Xinje XDPPro project, PLC1: XD3-32 (software 3.7.14 2021-12-24)

PROGRAM 梯形图

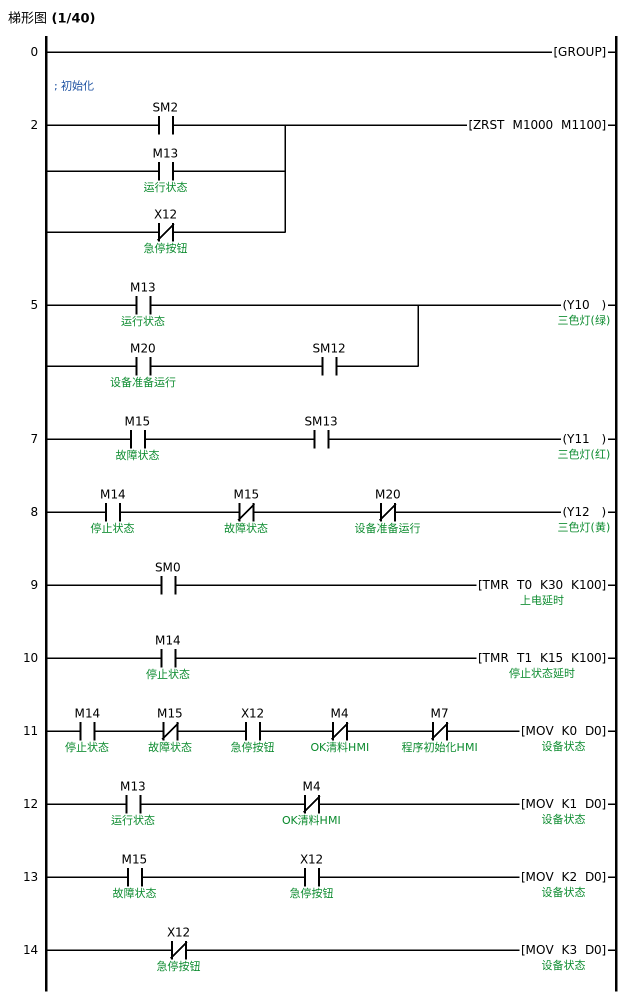
GROUP
; 初始化
LD     SM2
OR     M13	; 运行状态
ORI    X12	; 急停按钮
ZRST   M1000 M1100
LD     M13	; 运行状态
LD     M20	; 设备准备运行
AND    SM12
ORB
OUT    Y10	; 三色灯(绿)
LD     M15	; 故障状态
AND    SM13
OUT    Y11	; 三色灯(红)
LD     M14	; 停止状态
ANI    M15	; 故障状态
ANI    M20	; 设备准备运行
OUT    Y12	; 三色灯(黄)
LD     SM0
TMR    T0 K30 K100	; 上电延时
LD     M14	; 停止状态
TMR    T1 K15 K100	; 停止状态延时
LD     M14	; 停止状态
ANI    M15	; 故障状态
AND    X12	; 急停按钮
ANI    M4	; OK清料HMI
ANI    M7	; 程序初始化HMI
MOV    K0 D0	; 设备状态
LD     M13	; 运行状态
ANI    M4	; OK清料HMI
MOV    K1 D0	; 设备状态
LD     M15	; 故障状态
AND    X12	; 急停按钮
MOV    K2 D0	; 设备状态
LDI    X12	; 急停按钮
MOV    K3 D0	; 设备状态

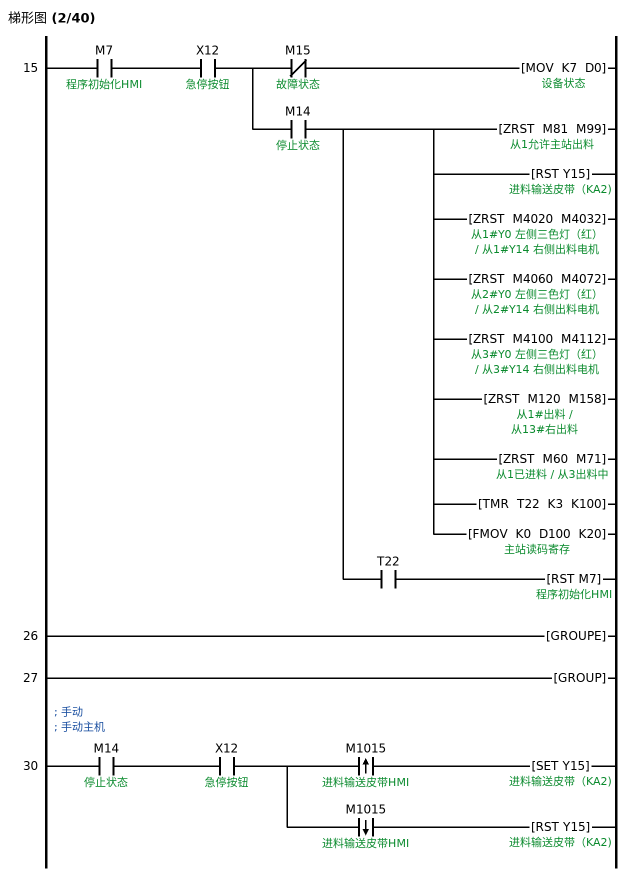
LD     M7	; 程序初始化HMI
AND    X12	; 急停按钮
MPS
ANI    M15	; 故障状态
MOV    K7 D0	; 设备状态
MPP
AND    M14	; 停止状态
ZRST   M81 M99	; 从1允许主站出料
RST    Y15	; 进料输送皮带（KA2)
ZRST   M4020 M4032	; 从1#Y0 左侧三色灯（红） / 从1#Y14 右侧出料电机
ZRST   M4060 M4072	; 从2#Y0 左侧三色灯（红） / 从2#Y14 右侧出料电机
ZRST   M4100 M4112	; 从3#Y0 左侧三色灯（红） / 从3#Y14 右侧出料电机
ZRST   M120 M158	; 从1#出料 / 从13#右出料
ZRST   M60 M71	; 从1已进料 / 从3出料中
TMR    T22 K3 K100
FMOV   K0 D100 K20	; 主站读码寄存
AND    T22
RST    M7	; 程序初始化HMI
GROUPE
GROUP
; 手动
; 手动主机
LD     M14	; 停止状态
AND    X12	; 急停按钮
MPS
ANDP   M1015	; 进料输送皮带HMI
SET    Y15	; 进料输送皮带（KA2)
MPP
ANDF   M1015	; 进料输送皮带HMI
RST    Y15	; 进料输送皮带（KA2)

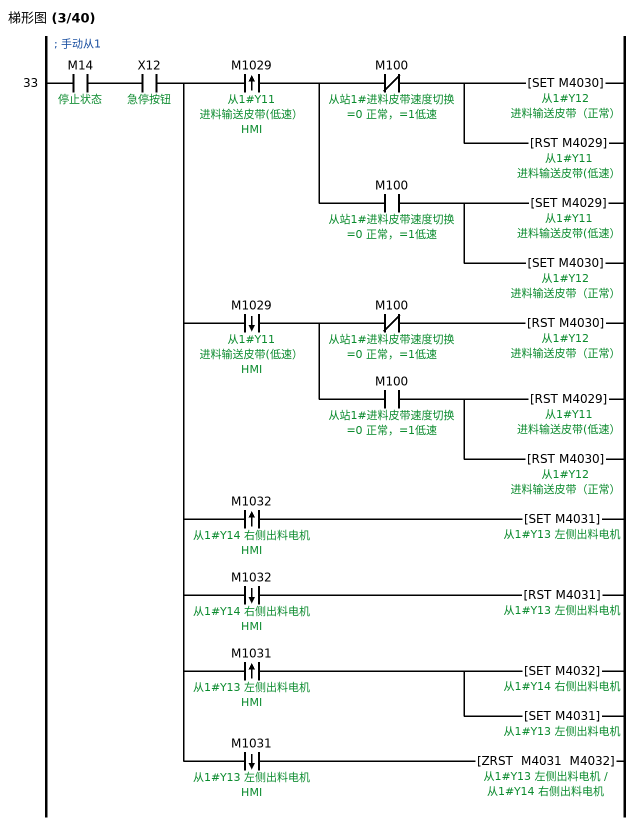
; 手动从1
LD     M14	; 停止状态
AND    X12	; 急停按钮
MPS
ANDP   M1029	; 从1#Y11 进料输送皮带(低速）       HMI
MPS
ANI    M100	; 从站1#进料皮带速度切换=0 正常，=1低速
SET    M4030	; 从1#Y12 进料输送皮带（正常）
RST    M4029	; 从1#Y11 进料输送皮带(低速）
MPP
AND    M100	; 从站1#进料皮带速度切换=0 正常，=1低速
SET    M4029	; 从1#Y11 进料输送皮带(低速）
SET    M4030	; 从1#Y12 进料输送皮带（正常）
MRD
ANDF   M1029	; 从1#Y11 进料输送皮带(低速）       HMI
MPS
ANI    M100	; 从站1#进料皮带速度切换=0 正常，=1低速
RST    M4030	; 从1#Y12 进料输送皮带（正常）
MPP
AND    M100	; 从站1#进料皮带速度切换=0 正常，=1低速
RST    M4029	; 从1#Y11 进料输送皮带(低速）
RST    M4030	; 从1#Y12 进料输送皮带（正常）
MRD
ANDP   M1032	; 从1#Y14 右侧出料电机       HMI
SET    M4031	; 从1#Y13 左侧出料电机
MRD
ANDF   M1032	; 从1#Y14 右侧出料电机       HMI
RST    M4031	; 从1#Y13 左侧出料电机
MRD
ANDP   M1031	; 从1#Y13 左侧出料电机       HMI
SET    M4032	; 从1#Y14 右侧出料电机
SET    M4031	; 从1#Y13 左侧出料电机
MPP
ANDF   M1031	; 从1#Y13 左侧出料电机       HMI
ZRST   M4031 M4032	; 从1#Y13 左侧出料电机 / 从1#Y14 右侧出料电机

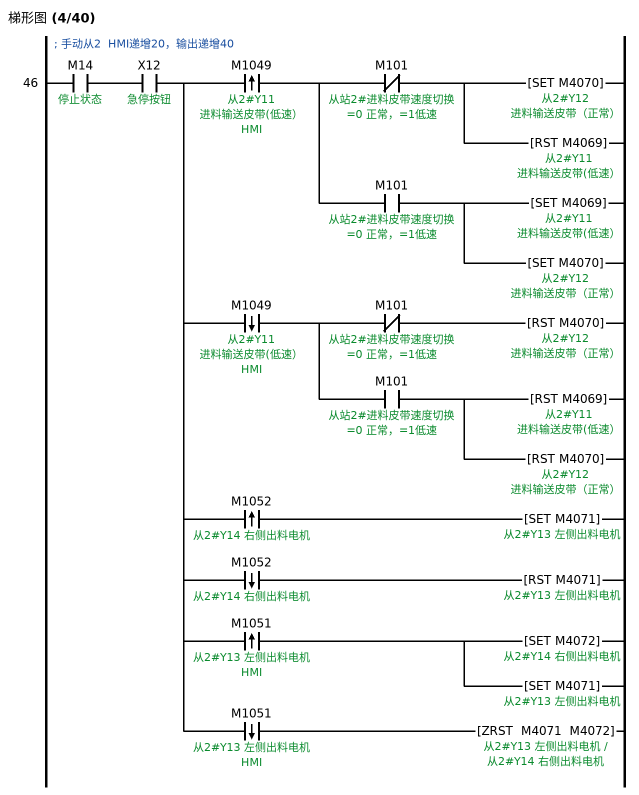
; 手动从2  HMI递增20，输出递增40
LD     M14	; 停止状态
AND    X12	; 急停按钮
MPS
ANDP   M1049	; 从2#Y11 进料输送皮带(低速）       HMI
MPS
ANI    M101	; 从站2#进料皮带速度切换=0 正常，=1低速
SET    M4070	; 从2#Y12 进料输送皮带（正常）
RST    M4069	; 从2#Y11 进料输送皮带(低速）
MPP
AND    M101	; 从站2#进料皮带速度切换=0 正常，=1低速
SET    M4069	; 从2#Y11 进料输送皮带(低速）
SET    M4070	; 从2#Y12 进料输送皮带（正常）
MRD
ANDF   M1049	; 从2#Y11 进料输送皮带(低速）       HMI
MPS
ANI    M101	; 从站2#进料皮带速度切换=0 正常，=1低速
RST    M4070	; 从2#Y12 进料输送皮带（正常）
MPP
AND    M101	; 从站2#进料皮带速度切换=0 正常，=1低速
RST    M4069	; 从2#Y11 进料输送皮带(低速）
RST    M4070	; 从2#Y12 进料输送皮带（正常）
MRD
ANDP   M1052	; 从2#Y14 右侧出料电机
SET    M4071	; 从2#Y13 左侧出料电机
MRD
ANDF   M1052	; 从2#Y14 右侧出料电机
RST    M4071	; 从2#Y13 左侧出料电机
MRD
ANDP   M1051	; 从2#Y13 左侧出料电机       HMI
SET    M4072	; 从2#Y14 右侧出料电机
SET    M4071	; 从2#Y13 左侧出料电机
MPP
ANDF   M1051	; 从2#Y13 左侧出料电机       HMI
ZRST   M4071 M4072	; 从2#Y13 左侧出料电机 / 从2#Y14 右侧出料电机

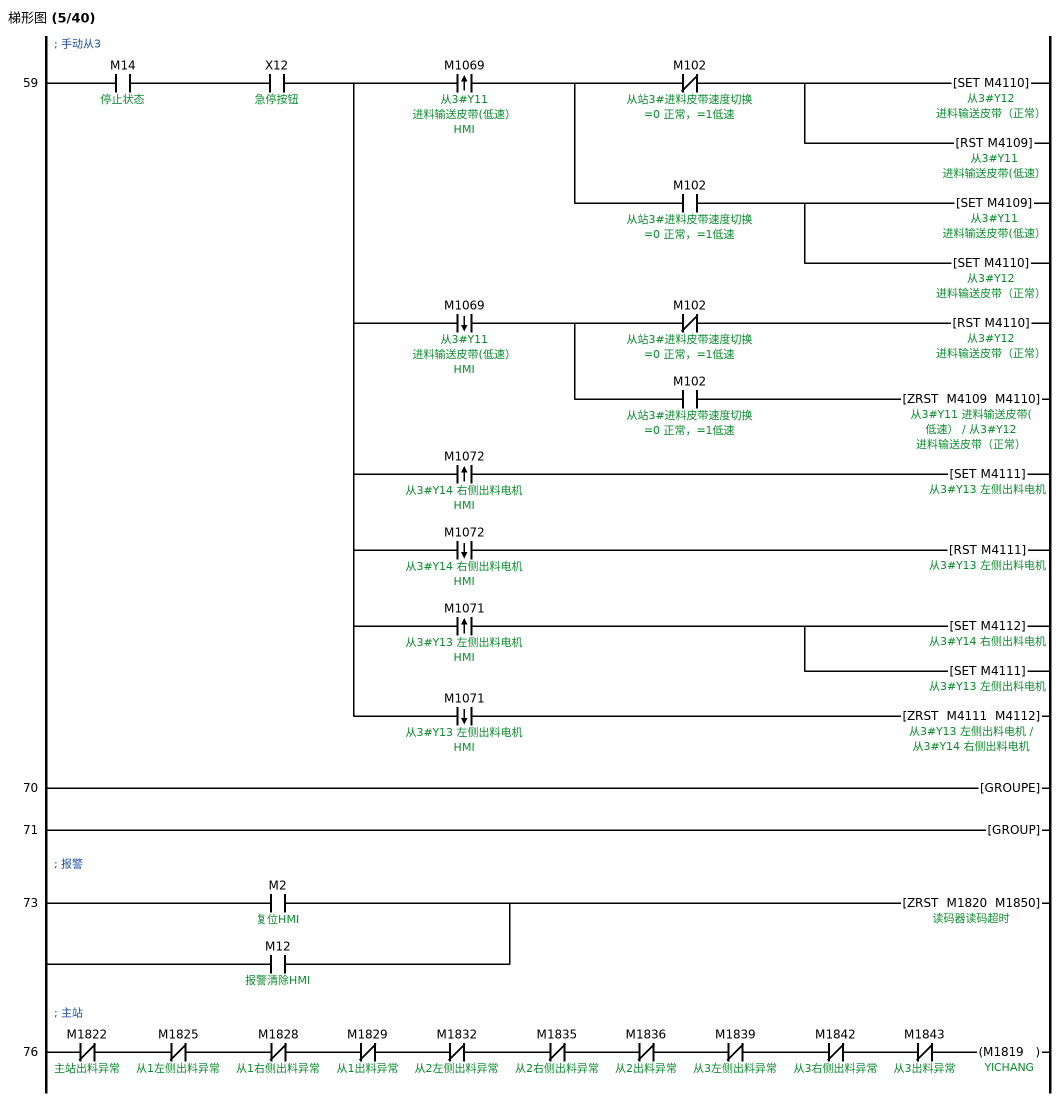
; 手动从3
LD     M14	; 停止状态
AND    X12	; 急停按钮
MPS
ANDP   M1069	; 从3#Y11 进料输送皮带(低速）       HMI
MPS
ANI    M102	; 从站3#进料皮带速度切换=0 正常，=1低速
SET    M4110	; 从3#Y12 进料输送皮带（正常）
RST    M4109	; 从3#Y11 进料输送皮带(低速）
MPP
AND    M102	; 从站3#进料皮带速度切换=0 正常，=1低速
SET    M4109	; 从3#Y11 进料输送皮带(低速）
SET    M4110	; 从3#Y12 进料输送皮带（正常）
MRD
ANDF   M1069	; 从3#Y11 进料输送皮带(低速）       HMI
MPS
ANI    M102	; 从站3#进料皮带速度切换=0 正常，=1低速
RST    M4110	; 从3#Y12 进料输送皮带（正常）
MPP
AND    M102	; 从站3#进料皮带速度切换=0 正常，=1低速
ZRST   M4109 M4110	; 从3#Y11 进料输送皮带(低速） / 从3#Y12 进料输送皮带（正常）
MRD
ANDP   M1072	; 从3#Y14 右侧出料电机       HMI
SET    M4111	; 从3#Y13 左侧出料电机
MRD
ANDF   M1072	; 从3#Y14 右侧出料电机       HMI
RST    M4111	; 从3#Y13 左侧出料电机
MRD
ANDP   M1071	; 从3#Y13 左侧出料电机       HMI
SET    M4112	; 从3#Y14 右侧出料电机
SET    M4111	; 从3#Y13 左侧出料电机
MPP
ANDF   M1071	; 从3#Y13 左侧出料电机       HMI
ZRST   M4111 M4112	; 从3#Y13 左侧出料电机 / 从3#Y14 右侧出料电机
GROUPE
GROUP
; 报警
LD     M2	; 复位HMI
OR     M12	; 报警清除HMI
ZRST   M1820 M1850	; 读码器读码超时
; 主站
LDI    M1822	; 主站出料异常
ANI    M1825	; 从1左侧出料异常
ANI    M1828	; 从1右侧出料异常
ANI    M1829	; 从1出料异常
ANI    M1832	; 从2左侧出料异常
ANI    M1835	; 从2右侧出料异常
ANI    M1836	; 从2出料异常
ANI    M1839	; 从3左侧出料异常
ANI    M1842	; 从3右侧出料异常
ANI    M1843	; 从3出料异常
OUT    M1819	; YICHANG

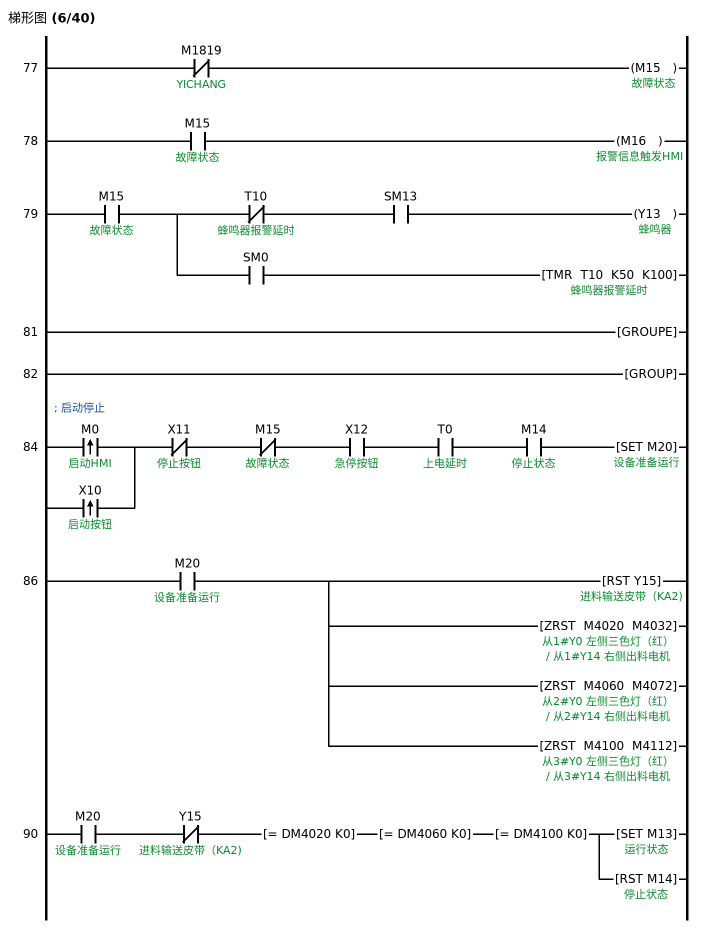
LDI    M1819	; YICHANG
OUT    M15	; 故障状态
LD     M15	; 故障状态
OUT    M16	; 报警信息触发HMI
LD     M15	; 故障状态
MPS
ANI    T10	; 蜂鸣器报警延时
AND    SM13
OUT    Y13	; 蜂鸣器
MPP
AND    SM0
TMR    T10 K50 K100	; 蜂鸣器报警延时
GROUPE
GROUP
; 启动停止
LDP    M0	; 启动HMI
ORP    X10	; 启动按钮
ANI    X11	; 停止按钮
ANI    M15	; 故障状态
AND    X12	; 急停按钮
AND    T0	; 上电延时
AND    M14	; 停止状态
SET    M20	; 设备准备运行
LD     M20	; 设备准备运行
RST    Y15	; 进料输送皮带（KA2)
ZRST   M4020 M4032	; 从1#Y0 左侧三色灯（红） / 从1#Y14 右侧出料电机
ZRST   M4060 M4072	; 从2#Y0 左侧三色灯（红） / 从2#Y14 右侧出料电机
ZRST   M4100 M4112	; 从3#Y0 左侧三色灯（红） / 从3#Y14 右侧出料电机
LD     M20	; 设备准备运行
ANI    Y15	; 进料输送皮带（KA2)
AND=   DM4020 K0
AND=   DM4060 K0
AND=   DM4100 K0
SET    M13	; 运行状态
RST    M14	; 停止状态

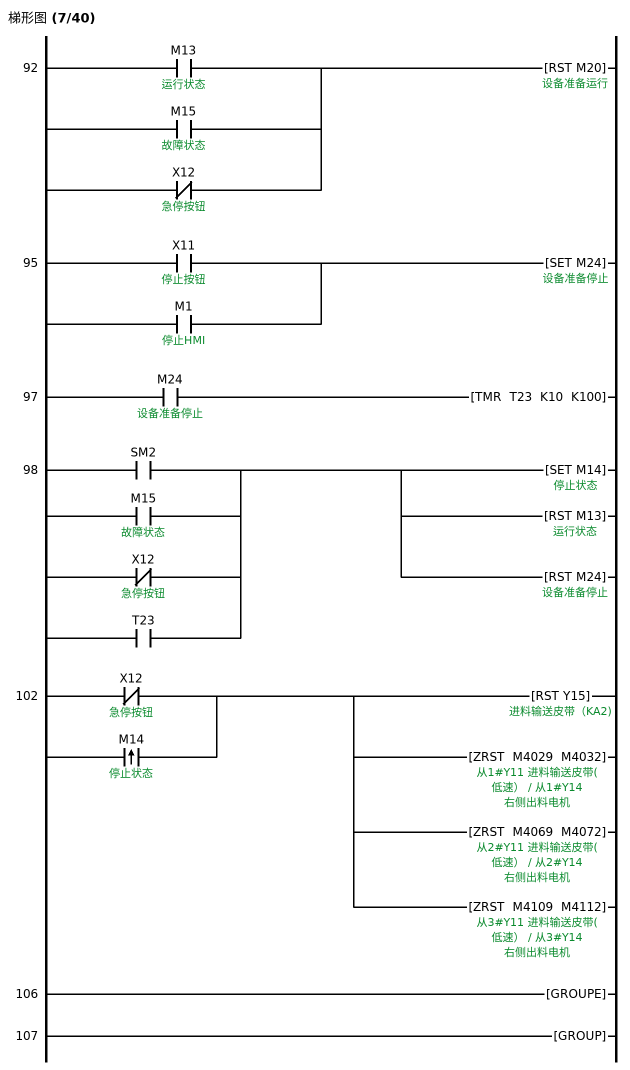
LD     M13	; 运行状态
OR     M15	; 故障状态
ORI    X12	; 急停按钮
RST    M20	; 设备准备运行
LD     X11	; 停止按钮
OR     M1	; 停止HMI
SET    M24	; 设备准备停止
LD     M24	; 设备准备停止
TMR    T23 K10 K100
LD     SM2
OR     M15	; 故障状态
ORI    X12	; 急停按钮
OR     T23
SET    M14	; 停止状态
RST    M13	; 运行状态
RST    M24	; 设备准备停止
LDI    X12	; 急停按钮
ORP    M14	; 停止状态
RST    Y15	; 进料输送皮带（KA2)
ZRST   M4029 M4032	; 从1#Y11 进料输送皮带(低速） / 从1#Y14 右侧出料电机
ZRST   M4069 M4072	; 从2#Y11 进料输送皮带(低速） / 从2#Y14 右侧出料电机
ZRST   M4109 M4112	; 从3#Y11 进料输送皮带(低速） / 从3#Y14 右侧出料电机
GROUPE
GROUP

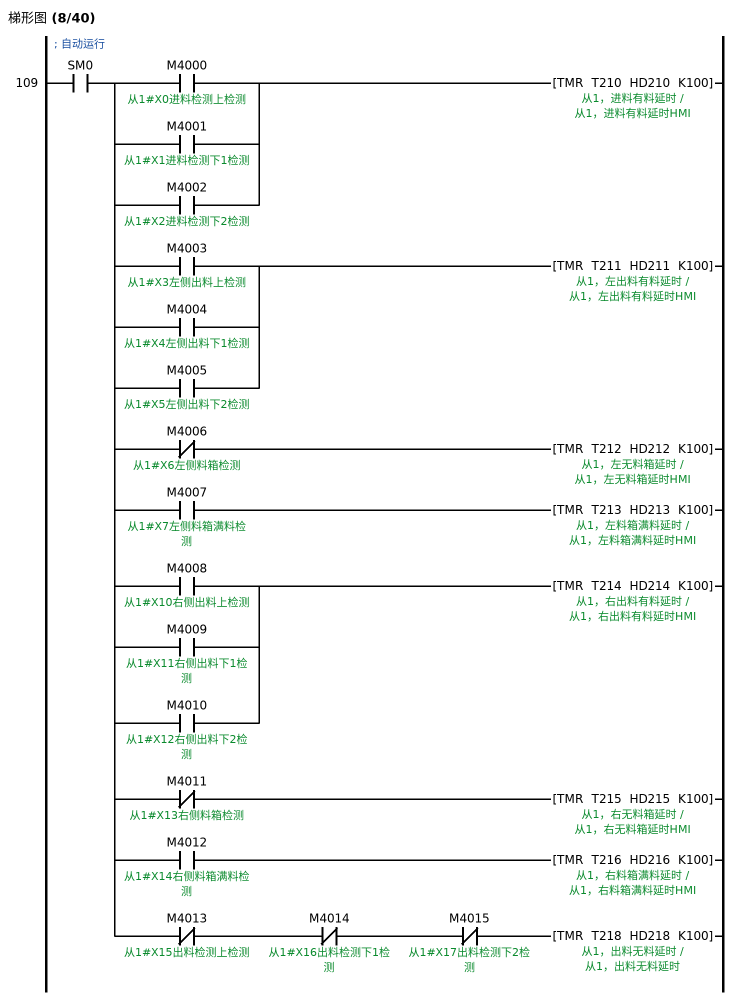
; 自动运行
LD     SM0
MPS
LD     M4000	; 从1#X0进料检测上检测
OR     M4001	; 从1#X1进料检测下1检测
OR     M4002	; 从1#X2进料检测下2检测
ANB
TMR    T210 HD210 K100	; 从1，进料有料延时 / 从1，进料有料延时HMI
MRD
LD     M4003	; 从1#X3左侧出料上检测
OR     M4004	; 从1#X4左侧出料下1检测
OR     M4005	; 从1#X5左侧出料下2检测
ANB
TMR    T211 HD211 K100	; 从1，左出料有料延时 / 从1，左出料有料延时HMI
MRD
ANI    M4006	; 从1#X6左侧料箱检测
TMR    T212 HD212 K100	; 从1，左无料箱延时 / 从1，左无料箱延时HMI
MRD
AND    M4007	; 从1#X7左侧料箱满料检测
TMR    T213 HD213 K100	; 从1，左料箱满料延时 / 从1，左料箱满料延时HMI
MRD
LD     M4008	; 从1#X10右侧出料上检测
OR     M4009	; 从1#X11右侧出料下1检测
OR     M4010	; 从1#X12右侧出料下2检测
ANB
TMR    T214 HD214 K100	; 从1，右出料有料延时 / 从1，右出料有料延时HMI
MRD
ANI    M4011	; 从1#X13右侧料箱检测
TMR    T215 HD215 K100	; 从1，右无料箱延时 / 从1，右无料箱延时HMI
MRD
AND    M4012	; 从1#X14右侧料箱满料检测
TMR    T216 HD216 K100	; 从1，右料箱满料延时 / 从1，右料箱满料延时HMI
MPP
ANI    M4013	; 从1#X15出料检测上检测
ANI    M4014	; 从1#X16出料检测下1检测
ANI    M4015	; 从1#X17出料检测下2检测
TMR    T218 HD218 K100	; 从1，出料无料延时 / 从1，出料无料延时

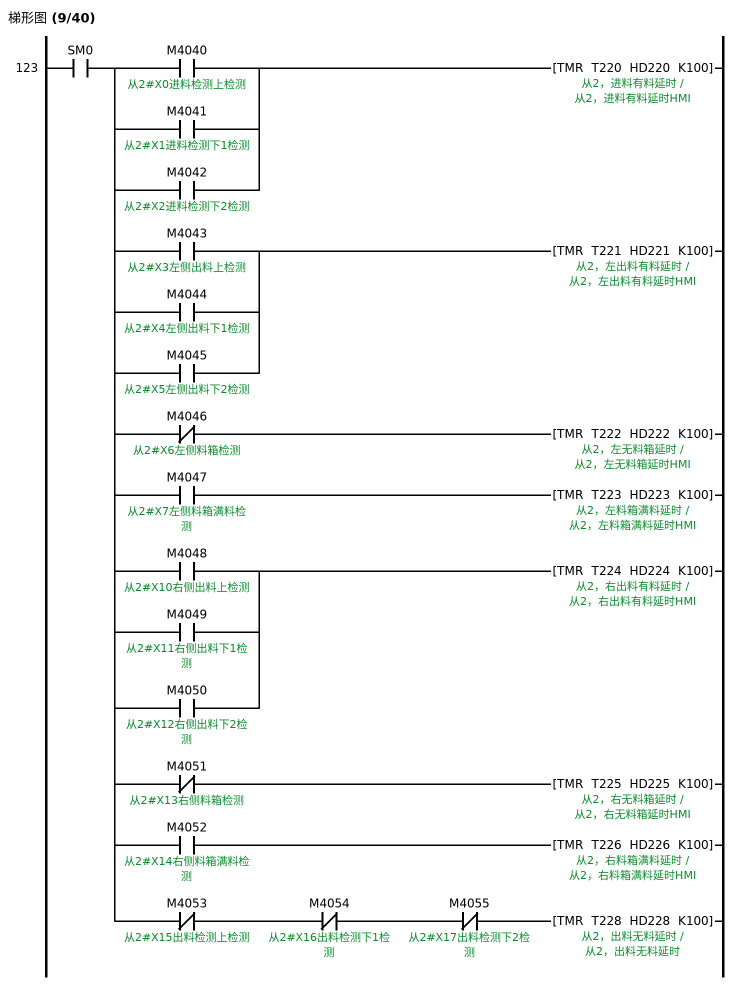
LD     SM0
MPS
LD     M4040	; 从2#X0进料检测上检测
OR     M4041	; 从2#X1进料检测下1检测
OR     M4042	; 从2#X2进料检测下2检测
ANB
TMR    T220 HD220 K100	; 从2，进料有料延时 / 从2，进料有料延时HMI
MRD
LD     M4043	; 从2#X3左侧出料上检测
OR     M4044	; 从2#X4左侧出料下1检测
OR     M4045	; 从2#X5左侧出料下2检测
ANB
TMR    T221 HD221 K100	; 从2，左出料有料延时 / 从2，左出料有料延时HMI
MRD
ANI    M4046	; 从2#X6左侧料箱检测
TMR    T222 HD222 K100	; 从2，左无料箱延时 / 从2，左无料箱延时HMI
MRD
AND    M4047	; 从2#X7左侧料箱满料检测
TMR    T223 HD223 K100	; 从2，左料箱满料延时 / 从2，左料箱满料延时HMI
MRD
LD     M4048	; 从2#X10右侧出料上检测
OR     M4049	; 从2#X11右侧出料下1检测
OR     M4050	; 从2#X12右侧出料下2检测
ANB
TMR    T224 HD224 K100	; 从2，右出料有料延时 / 从2，右出料有料延时HMI
MRD
ANI    M4051	; 从2#X13右侧料箱检测
TMR    T225 HD225 K100	; 从2，右无料箱延时 / 从2，右无料箱延时HMI
MRD
AND    M4052	; 从2#X14右侧料箱满料检测
TMR    T226 HD226 K100	; 从2，右料箱满料延时 / 从2，右料箱满料延时HMI
MPP
ANI    M4053	; 从2#X15出料检测上检测
ANI    M4054	; 从2#X16出料检测下1检测
ANI    M4055	; 从2#X17出料检测下2检测
TMR    T228 HD228 K100	; 从2，出料无料延时 / 从2，出料无料延时

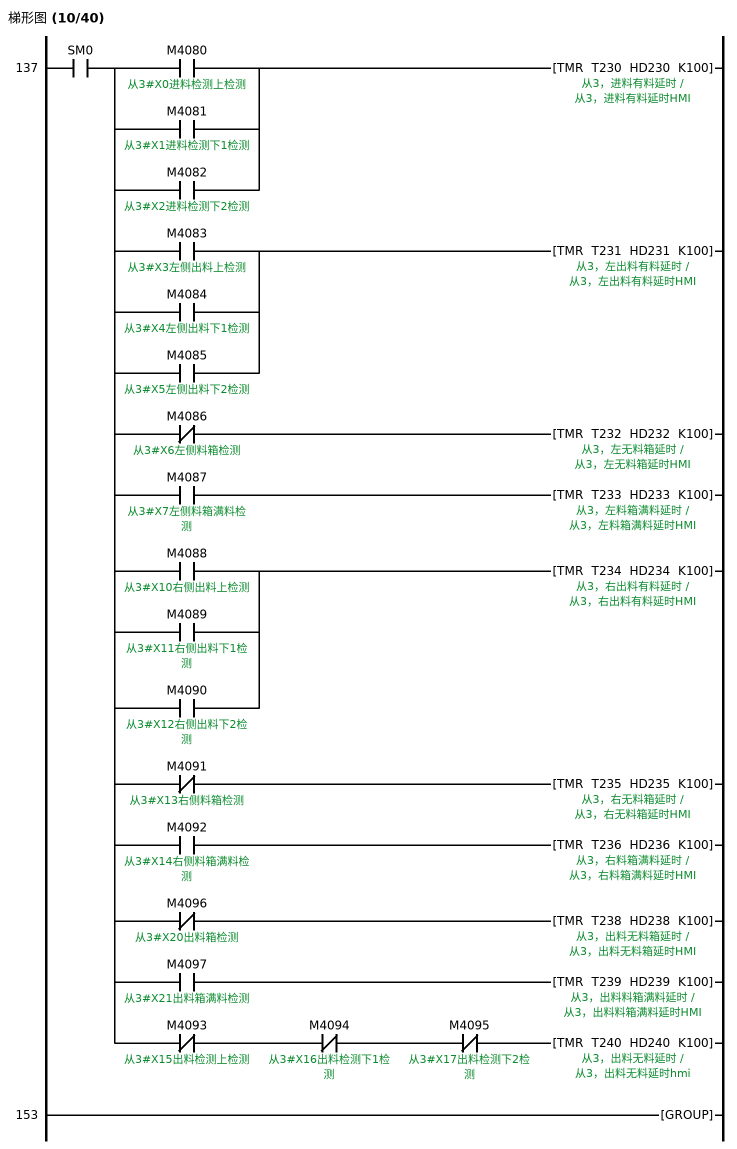
LD     SM0
MPS
LD     M4080	; 从3#X0进料检测上检测
OR     M4081	; 从3#X1进料检测下1检测
OR     M4082	; 从3#X2进料检测下2检测
ANB
TMR    T230 HD230 K100	; 从3，进料有料延时 / 从3，进料有料延时HMI
MRD
LD     M4083	; 从3#X3左侧出料上检测
OR     M4084	; 从3#X4左侧出料下1检测
OR     M4085	; 从3#X5左侧出料下2检测
ANB
TMR    T231 HD231 K100	; 从3，左出料有料延时 / 从3，左出料有料延时HMI
MRD
ANI    M4086	; 从3#X6左侧料箱检测
TMR    T232 HD232 K100	; 从3，左无料箱延时 / 从3，左无料箱延时HMI
MRD
AND    M4087	; 从3#X7左侧料箱满料检测
TMR    T233 HD233 K100	; 从3，左料箱满料延时 / 从3，左料箱满料延时HMI
MRD
LD     M4088	; 从3#X10右侧出料上检测
OR     M4089	; 从3#X11右侧出料下1检测
OR     M4090	; 从3#X12右侧出料下2检测
ANB
TMR    T234 HD234 K100	; 从3，右出料有料延时 / 从3，右出料有料延时HMI
MRD
ANI    M4091	; 从3#X13右侧料箱检测
TMR    T235 HD235 K100	; 从3，右无料箱延时 / 从3，右无料箱延时HMI
MRD
AND    M4092	; 从3#X14右侧料箱满料检测
TMR    T236 HD236 K100	; 从3，右料箱满料延时 / 从3，右料箱满料延时HMI
MRD
ANI    M4096	; 从3#X20出料箱检测
TMR    T238 HD238 K100	; 从3，出料无料箱延时 / 从3，出料无料箱延时HMI
MRD
AND    M4097	; 从3#X21出料箱满料检测
TMR    T239 HD239 K100	; 从3，出料料箱满料延时 / 从3，出料料箱满料延时HMI
MPP
ANI    M4093	; 从3#X15出料检测上检测
ANI    M4094	; 从3#X16出料检测下1检测
ANI    M4095	; 从3#X17出料检测下2检测
TMR    T240 HD240 K100	; 从3，出料无料延时 / 从3，出料无料延时hmi
GROUP

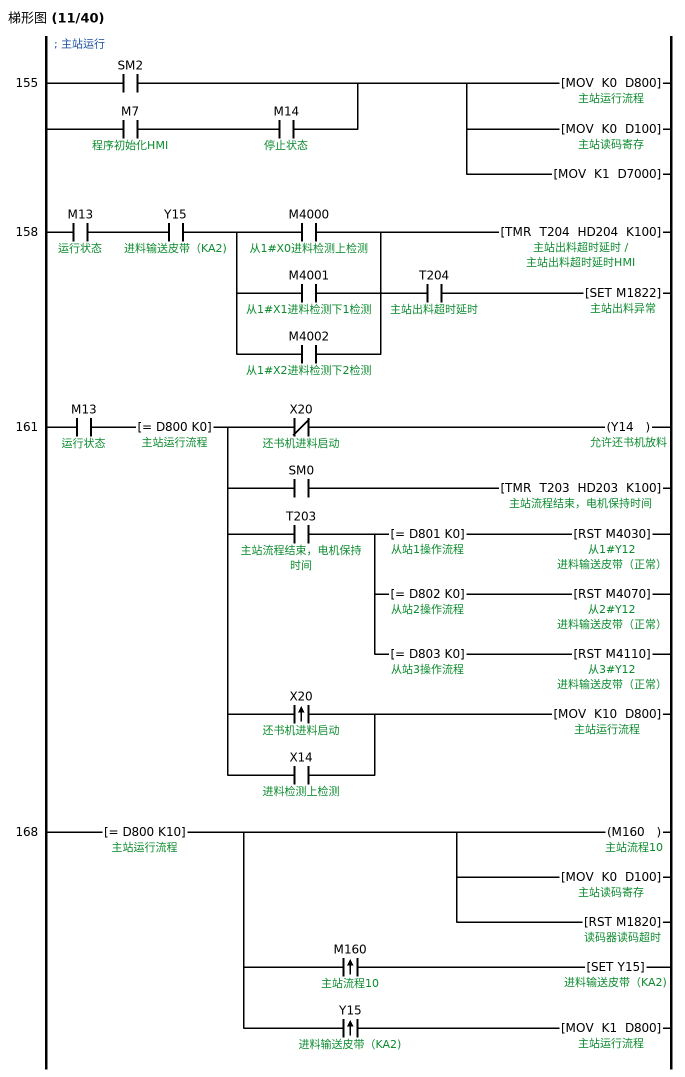
; 主站运行
LD     SM2
LD     M7	; 程序初始化HMI
AND    M14	; 停止状态
ORB
MOV    K0 D800	; 主站运行流程
MOV    K0 D100	; 主站读码寄存
MOV    K1 D7000
LD     M13	; 运行状态
AND    Y15	; 进料输送皮带（KA2)
LD     M4000	; 从1#X0进料检测上检测
OR     M4001	; 从1#X1进料检测下1检测
OR     M4002	; 从1#X2进料检测下2检测
ANB
TMR    T204 HD204 K100	; 主站出料超时延时 / 主站出料超时延时HMI
AND    T204	; 主站出料超时延时
SET    M1822	; 主站出料异常
LD     M13	; 运行状态
AND=   D800 K0	; 主站运行流程
MPS
ANI    X20	; 还书机进料启动
OUT    Y14	; 允许还书机放料
MRD
AND    SM0
TMR    T203 HD203 K100	; 主站流程结束，电机保持时间
MRD
AND    T203	; 主站流程结束，电机保持时间
MPS
AND=   D801 K0	; 从站1操作流程
RST    M4030	; 从1#Y12 进料输送皮带（正常）
MRD
AND=   D802 K0	; 从站2操作流程
RST    M4070	; 从2#Y12 进料输送皮带（正常）
MPP
AND=   D803 K0	; 从站3操作流程
RST    M4110	; 从3#Y12 进料输送皮带（正常）
MPP
LDP    X20	; 还书机进料启动
OR     X14	; 进料检测上检测
ANB
MOV    K10 D800	; 主站运行流程
LD=    D800 K10	; 主站运行流程
OUT    M160	; 主站流程10
MOV    K0 D100	; 主站读码寄存
RST    M1820	; 读码器读码超时
MPS
ANDP   M160	; 主站流程10
SET    Y15	; 进料输送皮带（KA2)
MPP
ANDP   Y15	; 进料输送皮带（KA2)
MOV    K1 D800	; 主站运行流程

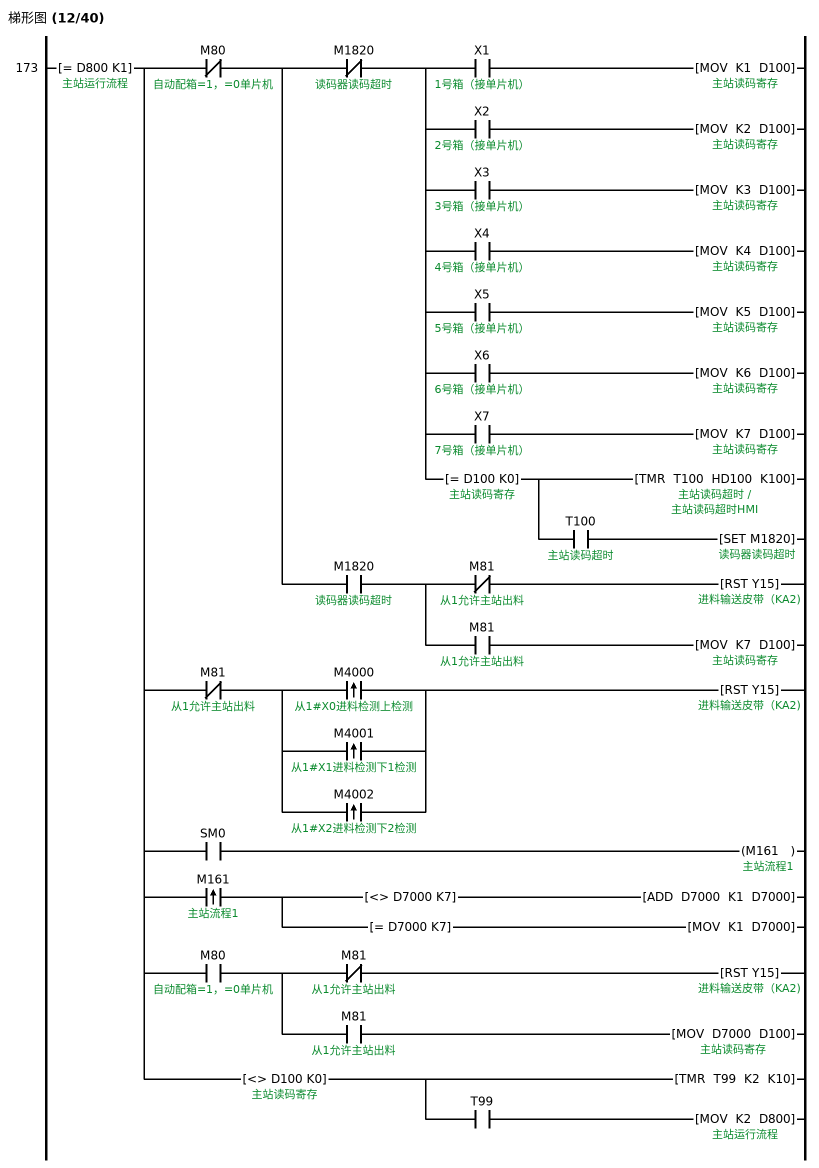
LD=    D800 K1	; 主站运行流程
MPS
ANI    M80	; 自动配箱=1，=0单片机
MPS
ANI    M1820	; 读码器读码超时
MPS
AND    X1	; 1号箱（接单片机）
MOV    K1 D100	; 主站读码寄存
MRD
AND    X2	; 2号箱（接单片机）
MOV    K2 D100	; 主站读码寄存
MRD
AND    X3	; 3号箱（接单片机）
MOV    K3 D100	; 主站读码寄存
MRD
AND    X4	; 4号箱（接单片机）
MOV    K4 D100	; 主站读码寄存
MRD
AND    X5	; 5号箱（接单片机）
MOV    K5 D100	; 主站读码寄存
MRD
AND    X6	; 6号箱（接单片机）
MOV    K6 D100	; 主站读码寄存
MRD
AND    X7	; 7号箱（接单片机）
MOV    K7 D100	; 主站读码寄存
MPP
AND=   D100 K0	; 主站读码寄存
TMR    T100 HD100 K100	; 主站读码超时 / 主站读码超时HMI
AND    T100	; 主站读码超时
SET    M1820	; 读码器读码超时
MPP
AND    M1820	; 读码器读码超时
MPS
ANI    M81	; 从1允许主站出料
RST    Y15	; 进料输送皮带（KA2)
MPP
AND    M81	; 从1允许主站出料
MOV    K7 D100	; 主站读码寄存
MRD
ANI    M81	; 从1允许主站出料
LDP    M4000	; 从1#X0进料检测上检测
ORP    M4001	; 从1#X1进料检测下1检测
ORP    M4002	; 从1#X2进料检测下2检测
ANB
RST    Y15	; 进料输送皮带（KA2)
MRD
AND    SM0
OUT    M161	; 主站流程1
MRD
ANDP   M161	; 主站流程1
MPS
AND<>  D7000 K7
ADD    D7000 K1 D7000
MPP
AND=   D7000 K7
MOV    K1 D7000
MRD
AND    M80	; 自动配箱=1，=0单片机
MPS
ANI    M81	; 从1允许主站出料
RST    Y15	; 进料输送皮带（KA2)
MPP
AND    M81	; 从1允许主站出料
MOV    D7000 D100	; 主站读码寄存
MPP
AND<>  D100 K0	; 主站读码寄存
TMR    T99 K2 K10
AND    T99
MOV    K2 D800	; 主站运行流程

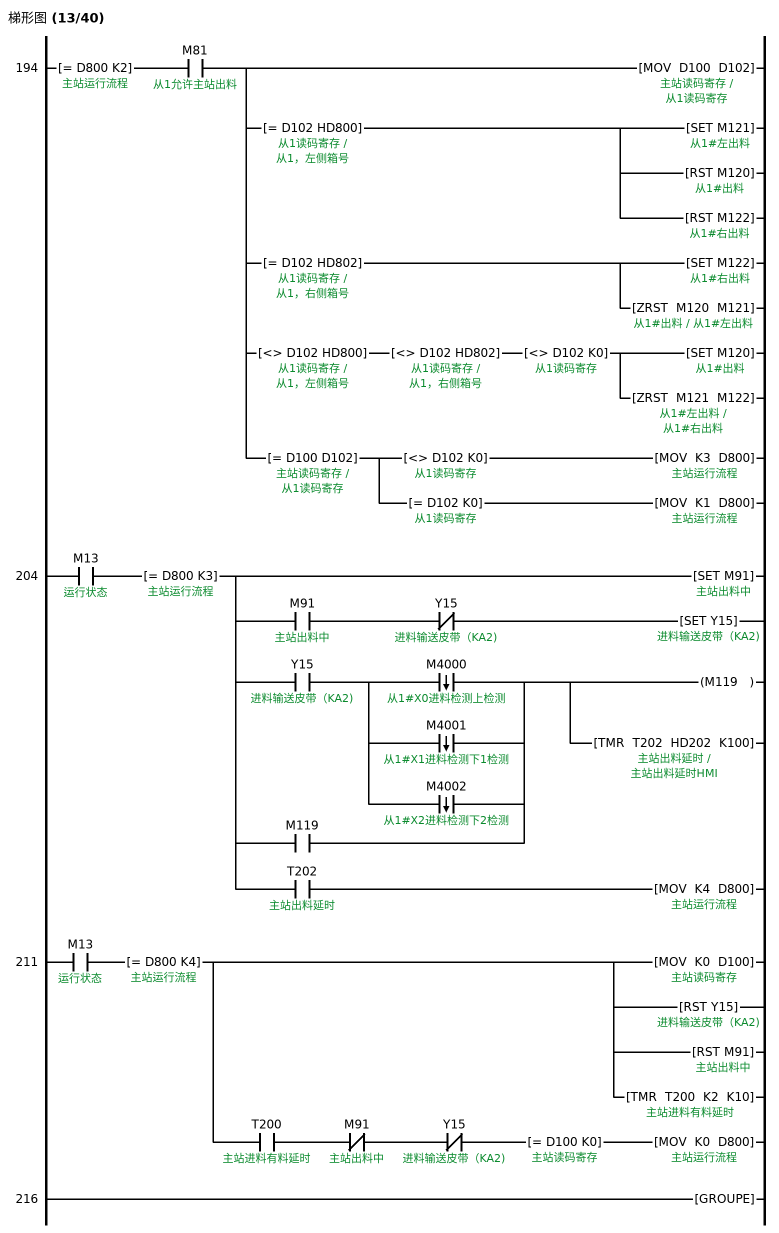
LD=    D800 K2	; 主站运行流程
AND    M81	; 从1允许主站出料
MOV    D100 D102	; 主站读码寄存 / 从1读码寄存
MPS
AND=   D102 HD800	; 从1读码寄存 / 从1，左侧箱号
SET    M121	; 从1#左出料
RST    M120	; 从1#出料
RST    M122	; 从1#右出料
MRD
AND=   D102 HD802	; 从1读码寄存 / 从1，右侧箱号
SET    M122	; 从1#右出料
ZRST   M120 M121	; 从1#出料 / 从1#左出料
MRD
AND<>  D102 HD800	; 从1读码寄存 / 从1，左侧箱号
AND<>  D102 HD802	; 从1读码寄存 / 从1，右侧箱号
AND<>  D102 K0	; 从1读码寄存
SET    M120	; 从1#出料
ZRST   M121 M122	; 从1#左出料 / 从1#右出料
MPP
AND=   D100 D102	; 主站读码寄存 / 从1读码寄存
MPS
AND<>  D102 K0	; 从1读码寄存
MOV    K3 D800	; 主站运行流程
MPP
AND=   D102 K0	; 从1读码寄存
MOV    K1 D800	; 主站运行流程
LD     M13	; 运行状态
AND=   D800 K3	; 主站运行流程
SET    M91	; 主站出料中
MPS
AND    M91	; 主站出料中
ANI    Y15	; 进料输送皮带（KA2)
SET    Y15	; 进料输送皮带（KA2)
MRD
LD     Y15	; 进料输送皮带（KA2)
LDF    M4000	; 从1#X0进料检测上检测
ORF    M4001	; 从1#X1进料检测下1检测
ORF    M4002	; 从1#X2进料检测下2检测
ANB
OR     M119
ANB
OUT    M119
TMR    T202 HD202 K100	; 主站出料延时 / 主站出料延时HMI
MPP
AND    T202	; 主站出料延时
MOV    K4 D800	; 主站运行流程
LD     M13	; 运行状态
AND=   D800 K4	; 主站运行流程
MOV    K0 D100	; 主站读码寄存
RST    Y15	; 进料输送皮带（KA2)
RST    M91	; 主站出料中
TMR    T200 K2 K10	; 主站进料有料延时
AND    T200	; 主站进料有料延时
ANI    M91	; 主站出料中
ANI    Y15	; 进料输送皮带（KA2)
AND=   D100 K0	; 主站读码寄存
MOV    K0 D800	; 主站运行流程
GROUPE

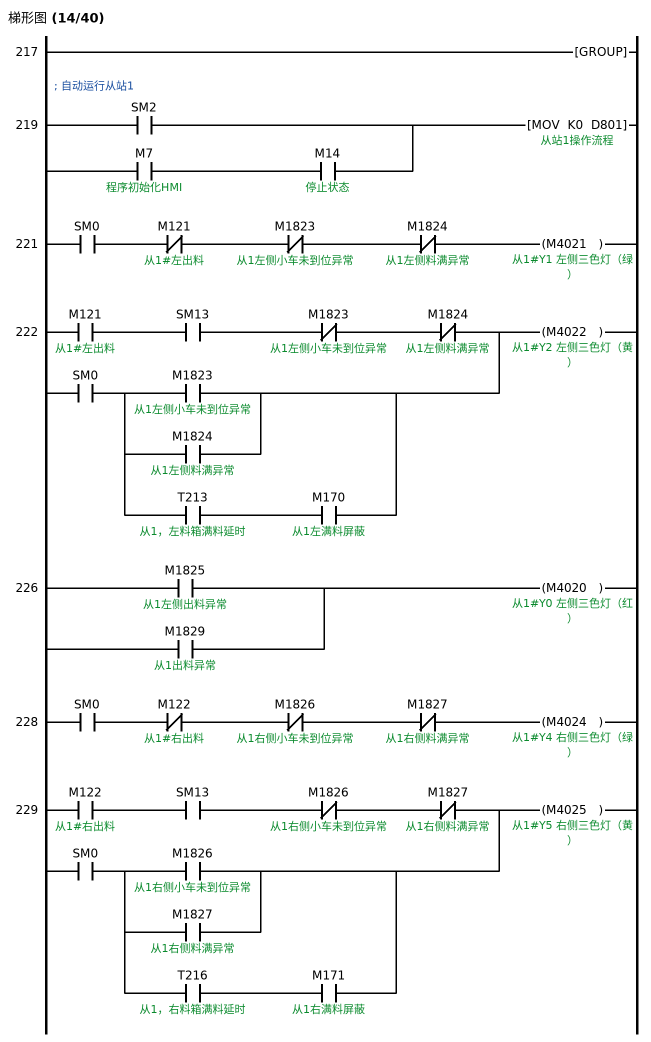
GROUP
; 自动运行从站1
LD     SM2
LD     M7	; 程序初始化HMI
AND    M14	; 停止状态
ORB
MOV    K0 D801	; 从站1操作流程
LD     SM0
ANI    M121	; 从1#左出料
ANI    M1823	; 从1左侧小车未到位异常
ANI    M1824	; 从1左侧料满异常
OUT    M4021	; 从1#Y1 左侧三色灯（绿）
LD     M121	; 从1#左出料
AND    SM13
ANI    M1823	; 从1左侧小车未到位异常
ANI    M1824	; 从1左侧料满异常
LD     SM0
LD     M1823	; 从1左侧小车未到位异常
OR     M1824	; 从1左侧料满异常
LD     T213	; 从1，左料箱满料延时
AND    M170	; 从1左满料屏蔽
ORB
ANB
ORB
OUT    M4022	; 从1#Y2 左侧三色灯（黄）
LD     M1825	; 从1左侧出料异常
OR     M1829	; 从1出料异常
OUT    M4020	; 从1#Y0 左侧三色灯（红）
LD     SM0
ANI    M122	; 从1#右出料
ANI    M1826	; 从1右侧小车未到位异常
ANI    M1827	; 从1右侧料满异常
OUT    M4024	; 从1#Y4 右侧三色灯（绿）
LD     M122	; 从1#右出料
AND    SM13
ANI    M1826	; 从1右侧小车未到位异常
ANI    M1827	; 从1右侧料满异常
LD     SM0
LD     M1826	; 从1右侧小车未到位异常
OR     M1827	; 从1右侧料满异常
LD     T216	; 从1，右料箱满料延时
AND    M171	; 从1右满料屏蔽
ORB
ANB
ORB
OUT    M4025	; 从1#Y5 右侧三色灯（黄）

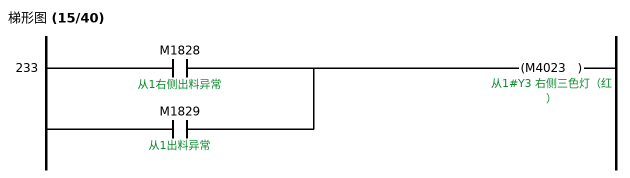
LD     M1828	; 从1右侧出料异常
OR     M1829	; 从1出料异常
OUT    M4023	; 从1#Y3 右侧三色灯（红）

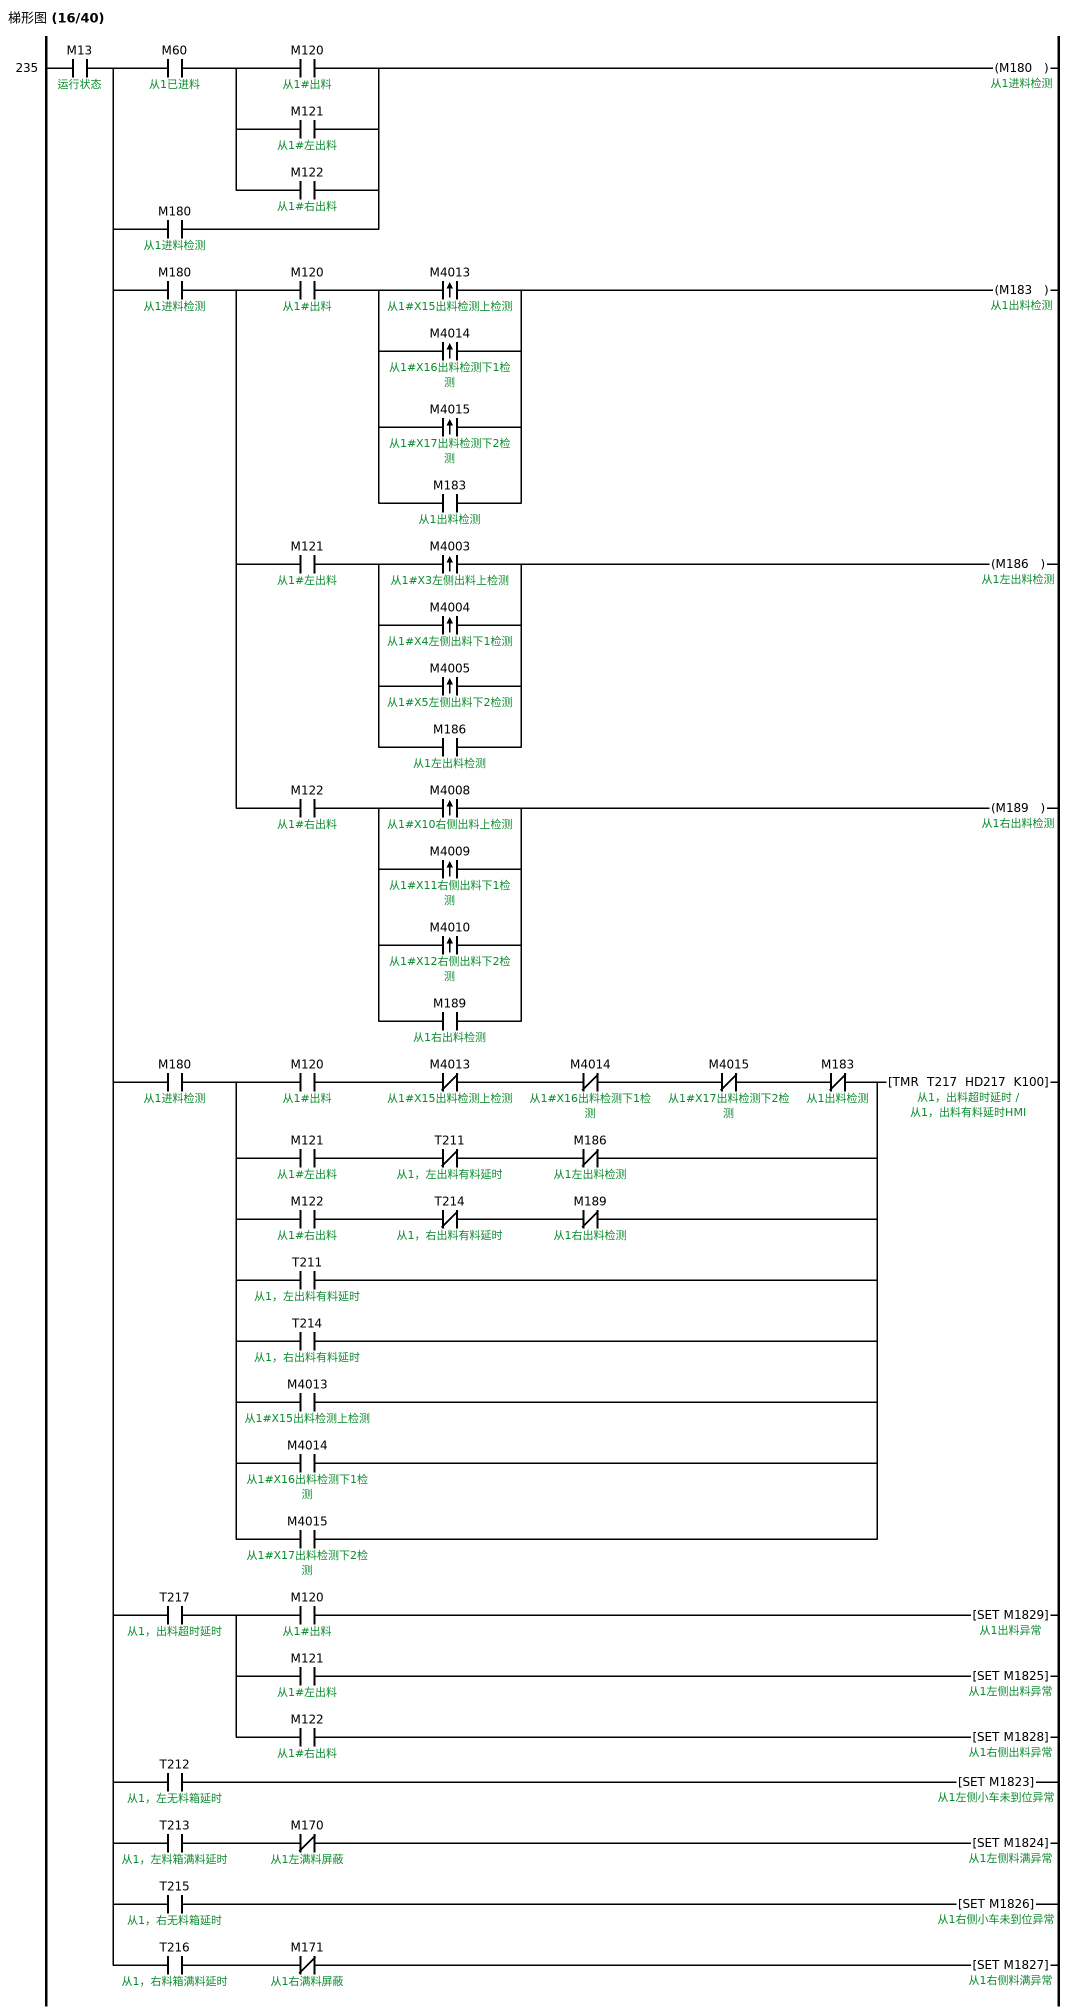
LD     M13	; 运行状态
MPS
LD     M60	; 从1已进料
LD     M120	; 从1#出料
OR     M121	; 从1#左出料
OR     M122	; 从1#右出料
ANB
OR     M180	; 从1进料检测
ANB
OUT    M180	; 从1进料检测
MRD
AND    M180	; 从1进料检测
MPS
AND    M120	; 从1#出料
LDP    M4013	; 从1#X15出料检测上检测
ORP    M4014	; 从1#X16出料检测下1检测
ORP    M4015	; 从1#X17出料检测下2检测
OR     M183	; 从1出料检测
ANB
OUT    M183	; 从1出料检测
MRD
AND    M121	; 从1#左出料
LDP    M4003	; 从1#X3左侧出料上检测
ORP    M4004	; 从1#X4左侧出料下1检测
ORP    M4005	; 从1#X5左侧出料下2检测
OR     M186	; 从1左出料检测
ANB
OUT    M186	; 从1左出料检测
MPP
AND    M122	; 从1#右出料
LDP    M4008	; 从1#X10右侧出料上检测
ORP    M4009	; 从1#X11右侧出料下1检测
ORP    M4010	; 从1#X12右侧出料下2检测
OR     M189	; 从1右出料检测
ANB
OUT    M189	; 从1右出料检测
MRD
AND    M180	; 从1进料检测
LD     M120	; 从1#出料
ANI    M4013	; 从1#X15出料检测上检测
ANI    M4014	; 从1#X16出料检测下1检测
ANI    M4015	; 从1#X17出料检测下2检测
ANI    M183	; 从1出料检测
LD     M121	; 从1#左出料
ANI    T211	; 从1，左出料有料延时
ANI    M186	; 从1左出料检测
ORB
LD     M122	; 从1#右出料
ANI    T214	; 从1，右出料有料延时
ANI    M189	; 从1右出料检测
ORB
OR     T211	; 从1，左出料有料延时
OR     T214	; 从1，右出料有料延时
OR     M4013	; 从1#X15出料检测上检测
OR     M4014	; 从1#X16出料检测下1检测
OR     M4015	; 从1#X17出料检测下2检测
ANB
TMR    T217 HD217 K100	; 从1，出料超时延时 / 从1，出料有料延时HMI
MRD
AND    T217	; 从1，出料超时延时
MPS
AND    M120	; 从1#出料
SET    M1829	; 从1出料异常
MRD
AND    M121	; 从1#左出料
SET    M1825	; 从1左侧出料异常
MPP
AND    M122	; 从1#右出料
SET    M1828	; 从1右侧出料异常
MRD
AND    T212	; 从1，左无料箱延时
SET    M1823	; 从1左侧小车未到位异常
MRD
AND    T213	; 从1，左料箱满料延时
ANI    M170	; 从1左满料屏蔽
SET    M1824	; 从1左侧料满异常
MRD
AND    T215	; 从1，右无料箱延时
SET    M1826	; 从1右侧小车未到位异常
MPP
AND    T216	; 从1，右料箱满料延时
ANI    M171	; 从1右满料屏蔽
SET    M1827	; 从1右侧料满异常

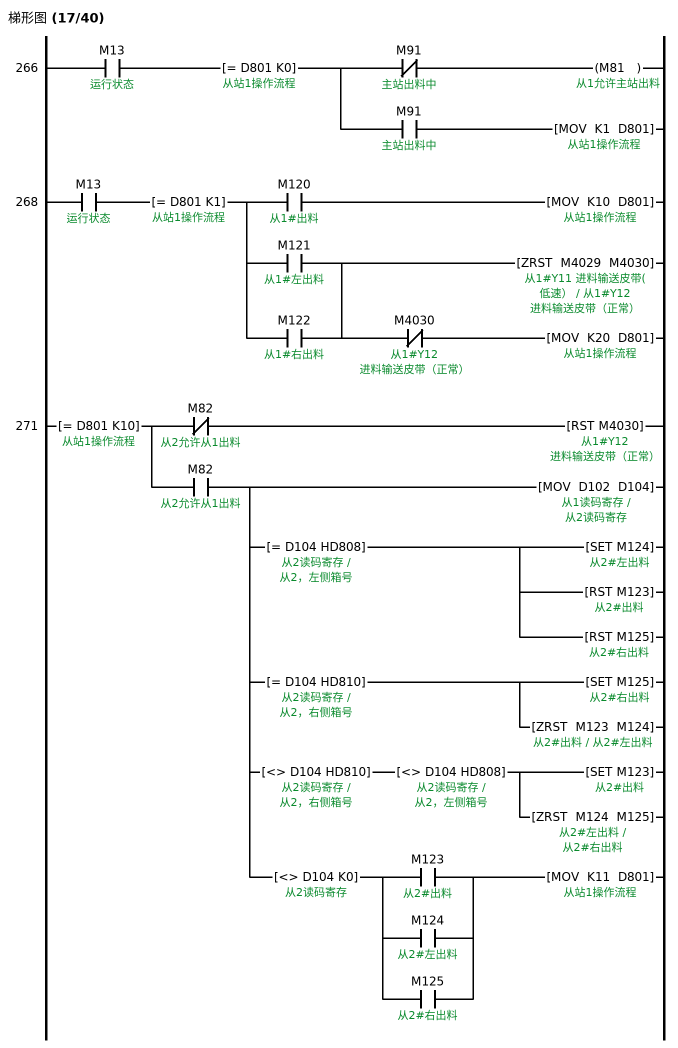
LD     M13	; 运行状态
AND=   D801 K0	; 从站1操作流程
MPS
ANI    M91	; 主站出料中
OUT    M81	; 从1允许主站出料
MPP
AND    M91	; 主站出料中
MOV    K1 D801	; 从站1操作流程
LD     M13	; 运行状态
AND=   D801 K1	; 从站1操作流程
MPS
AND    M120	; 从1#出料
MOV    K10 D801	; 从站1操作流程
MPP
LD     M121	; 从1#左出料
OR     M122	; 从1#右出料
ANB
ZRST   M4029 M4030	; 从1#Y11 进料输送皮带(低速） / 从1#Y12 进料输送皮带（正常）
ANI    M4030	; 从1#Y12 进料输送皮带（正常）
MOV    K20 D801	; 从站1操作流程
LD=    D801 K10	; 从站1操作流程
MPS
ANI    M82	; 从2允许从1出料
RST    M4030	; 从1#Y12 进料输送皮带（正常）
MPP
AND    M82	; 从2允许从1出料
MOV    D102 D104	; 从1读码寄存 / 从2读码寄存
MPS
AND=   D104 HD808	; 从2读码寄存 / 从2，左侧箱号
SET    M124	; 从2#左出料
RST    M123	; 从2#出料
RST    M125	; 从2#右出料
MRD
AND=   D104 HD810	; 从2读码寄存 / 从2，右侧箱号
SET    M125	; 从2#右出料
ZRST   M123 M124	; 从2#出料 / 从2#左出料
MRD
AND<>  D104 HD810	; 从2读码寄存 / 从2，右侧箱号
AND<>  D104 HD808	; 从2读码寄存 / 从2，左侧箱号
SET    M123	; 从2#出料
ZRST   M124 M125	; 从2#左出料 / 从2#右出料
MPP
AND<>  D104 K0	; 从2读码寄存
LD     M123	; 从2#出料
OR     M124	; 从2#左出料
OR     M125	; 从2#右出料
ANB
MOV    K11 D801	; 从站1操作流程

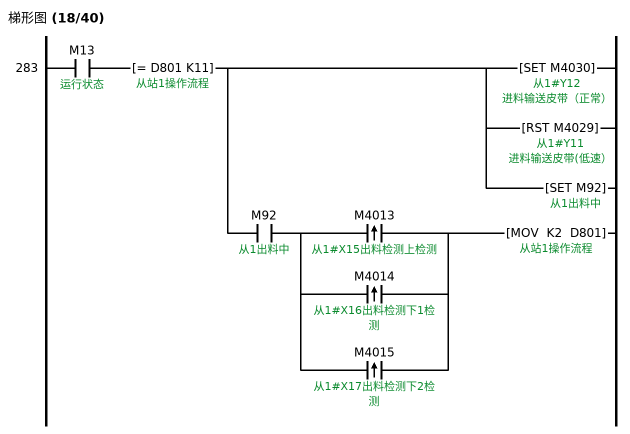
LD     M13	; 运行状态
AND=   D801 K11	; 从站1操作流程
SET    M4030	; 从1#Y12 进料输送皮带（正常）
RST    M4029	; 从1#Y11 进料输送皮带(低速）
SET    M92	; 从1出料中
AND    M92	; 从1出料中
LDP    M4013	; 从1#X15出料检测上检测
ORP    M4014	; 从1#X16出料检测下1检测
ORP    M4015	; 从1#X17出料检测下2检测
ANB
MOV    K2 D801	; 从站1操作流程

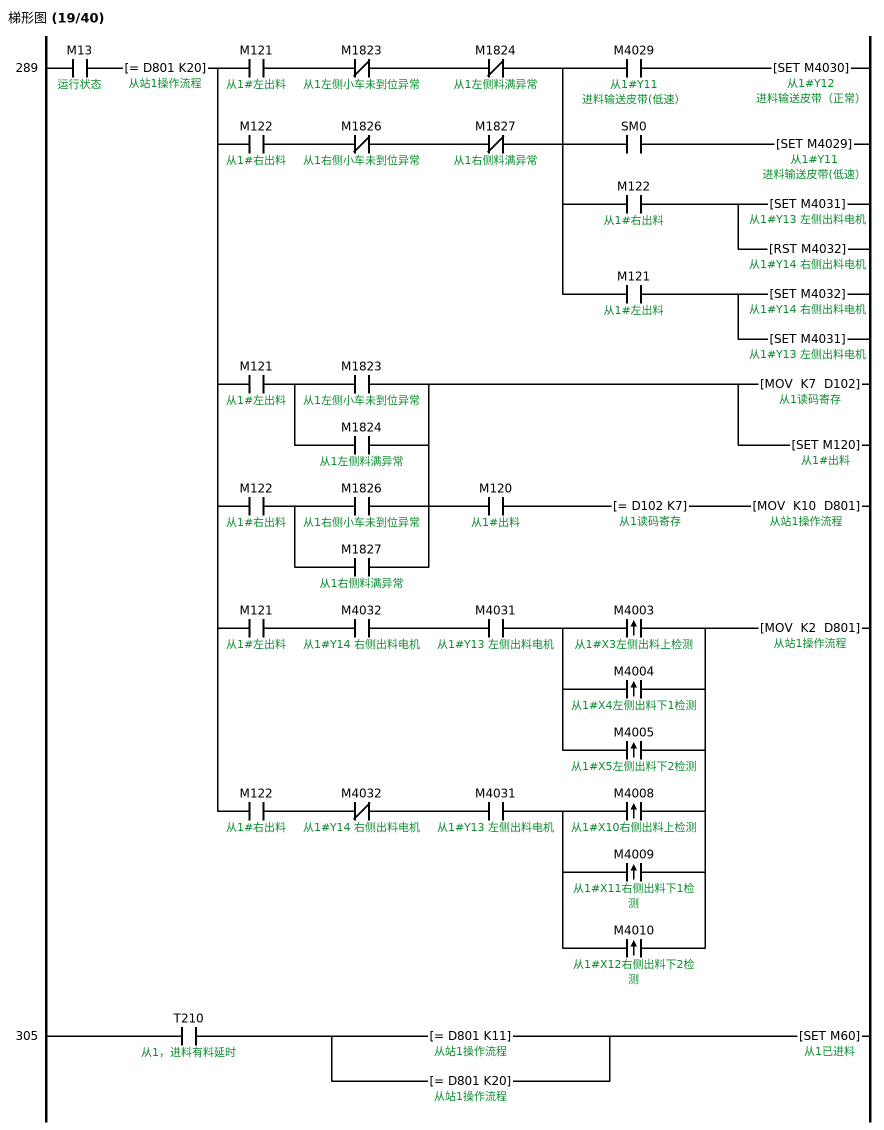
LD     M13	; 运行状态
AND=   D801 K20	; 从站1操作流程
MPS
LD     M121	; 从1#左出料
ANI    M1823	; 从1左侧小车未到位异常
ANI    M1824	; 从1左侧料满异常
LD     M122	; 从1#右出料
ANI    M1826	; 从1右侧小车未到位异常
ANI    M1827	; 从1右侧料满异常
ORB
ANB
MPS
AND    M4029	; 从1#Y11 进料输送皮带(低速）
SET    M4030	; 从1#Y12 进料输送皮带（正常）
MRD
AND    SM0
SET    M4029	; 从1#Y11 进料输送皮带(低速）
MRD
AND    M122	; 从1#右出料
SET    M4031	; 从1#Y13 左侧出料电机
RST    M4032	; 从1#Y14 右侧出料电机
MPP
AND    M121	; 从1#左出料
SET    M4032	; 从1#Y14 右侧出料电机
SET    M4031	; 从1#Y13 左侧出料电机
MRD
LD     M121	; 从1#左出料
LD     M1823	; 从1左侧小车未到位异常
OR     M1824	; 从1左侧料满异常
ANB
LD     M122	; 从1#右出料
LD     M1826	; 从1右侧小车未到位异常
OR     M1827	; 从1右侧料满异常
ANB
ORB
ANB
MOV    K7 D102	; 从1读码寄存
SET    M120	; 从1#出料
AND    M120	; 从1#出料
AND=   D102 K7	; 从1读码寄存
MOV    K10 D801	; 从站1操作流程
MPP
LD     M121	; 从1#左出料
AND    M4032	; 从1#Y14 右侧出料电机
AND    M4031	; 从1#Y13 左侧出料电机
LDP    M4003	; 从1#X3左侧出料上检测
ORP    M4004	; 从1#X4左侧出料下1检测
ORP    M4005	; 从1#X5左侧出料下2检测
ANB
LD     M122	; 从1#右出料
ANI    M4032	; 从1#Y14 右侧出料电机
AND    M4031	; 从1#Y13 左侧出料电机
LDP    M4008	; 从1#X10右侧出料上检测
ORP    M4009	; 从1#X11右侧出料下1检测
ORP    M4010	; 从1#X12右侧出料下2检测
ANB
ORB
ANB
MOV    K2 D801	; 从站1操作流程
LD     T210	; 从1，进料有料延时
LD=    D801 K11	; 从站1操作流程
OR=    D801 K20	; 从站1操作流程
ANB
SET    M60	; 从1已进料

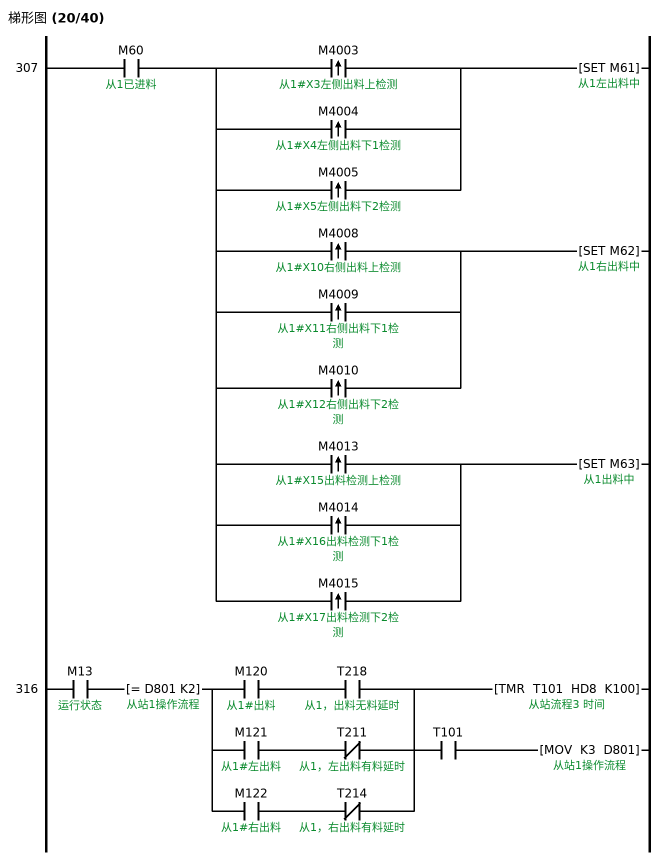
LD     M60	; 从1已进料
MPS
LDP    M4003	; 从1#X3左侧出料上检测
ORP    M4004	; 从1#X4左侧出料下1检测
ORP    M4005	; 从1#X5左侧出料下2检测
ANB
SET    M61	; 从1左出料中
MRD
LDP    M4008	; 从1#X10右侧出料上检测
ORP    M4009	; 从1#X11右侧出料下1检测
ORP    M4010	; 从1#X12右侧出料下2检测
ANB
SET    M62	; 从1右出料中
MPP
LDP    M4013	; 从1#X15出料检测上检测
ORP    M4014	; 从1#X16出料检测下1检测
ORP    M4015	; 从1#X17出料检测下2检测
ANB
SET    M63	; 从1出料中
LD     M13	; 运行状态
AND=   D801 K2	; 从站1操作流程
LD     M120	; 从1#出料
AND    T218	; 从1，出料无料延时
LD     M121	; 从1#左出料
ANI    T211	; 从1，左出料有料延时
ORB
LD     M122	; 从1#右出料
ANI    T214	; 从1，右出料有料延时
ORB
ANB
TMR    T101 HD8 K100	; 从站流程3 时间
AND    T101
MOV    K3 D801	; 从站1操作流程

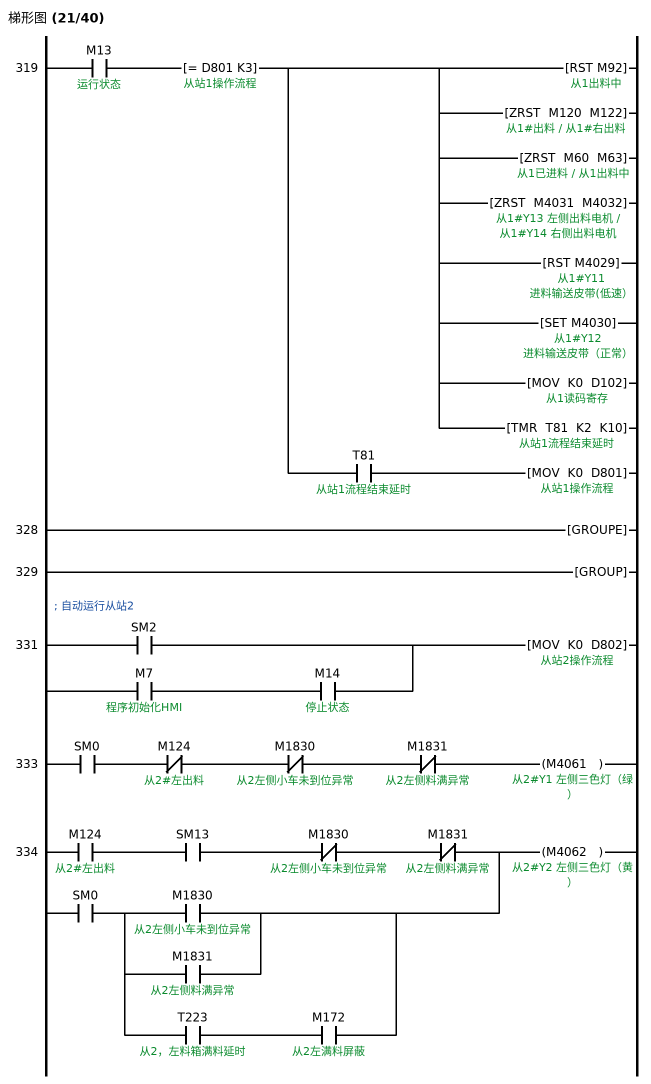
LD     M13	; 运行状态
AND=   D801 K3	; 从站1操作流程
RST    M92	; 从1出料中
ZRST   M120 M122	; 从1#出料 / 从1#右出料
ZRST   M60 M63	; 从1已进料 / 从1出料中
ZRST   M4031 M4032	; 从1#Y13 左侧出料电机 / 从1#Y14 右侧出料电机
RST    M4029	; 从1#Y11 进料输送皮带(低速）
SET    M4030	; 从1#Y12 进料输送皮带（正常）
MOV    K0 D102	; 从1读码寄存
TMR    T81 K2 K10	; 从站1流程结束延时
AND    T81	; 从站1流程结束延时
MOV    K0 D801	; 从站1操作流程
GROUPE
GROUP
; 自动运行从站2
LD     SM2
LD     M7	; 程序初始化HMI
AND    M14	; 停止状态
ORB
MOV    K0 D802	; 从站2操作流程
LD     SM0
ANI    M124	; 从2#左出料
ANI    M1830	; 从2左侧小车未到位异常
ANI    M1831	; 从2左侧料满异常
OUT    M4061	; 从2#Y1 左侧三色灯（绿）
LD     M124	; 从2#左出料
AND    SM13
ANI    M1830	; 从2左侧小车未到位异常
ANI    M1831	; 从2左侧料满异常
LD     SM0
LD     M1830	; 从2左侧小车未到位异常
OR     M1831	; 从2左侧料满异常
LD     T223	; 从2，左料箱满料延时
AND    M172	; 从2左满料屏蔽
ORB
ANB
ORB
OUT    M4062	; 从2#Y2 左侧三色灯（黄）

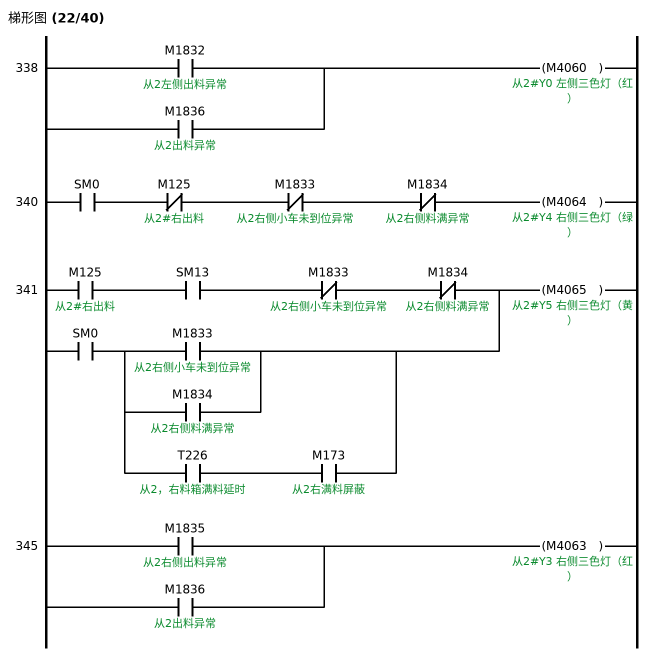
LD     M1832	; 从2左侧出料异常
OR     M1836	; 从2出料异常
OUT    M4060	; 从2#Y0 左侧三色灯（红）
LD     SM0
ANI    M125	; 从2#右出料
ANI    M1833	; 从2右侧小车未到位异常
ANI    M1834	; 从2右侧料满异常
OUT    M4064	; 从2#Y4 右侧三色灯（绿）
LD     M125	; 从2#右出料
AND    SM13
ANI    M1833	; 从2右侧小车未到位异常
ANI    M1834	; 从2右侧料满异常
LD     SM0
LD     M1833	; 从2右侧小车未到位异常
OR     M1834	; 从2右侧料满异常
LD     T226	; 从2，右料箱满料延时
AND    M173	; 从2右满料屏蔽
ORB
ANB
ORB
OUT    M4065	; 从2#Y5 右侧三色灯（黄）
LD     M1835	; 从2右侧出料异常
OR     M1836	; 从2出料异常
OUT    M4063	; 从2#Y3 右侧三色灯（红）

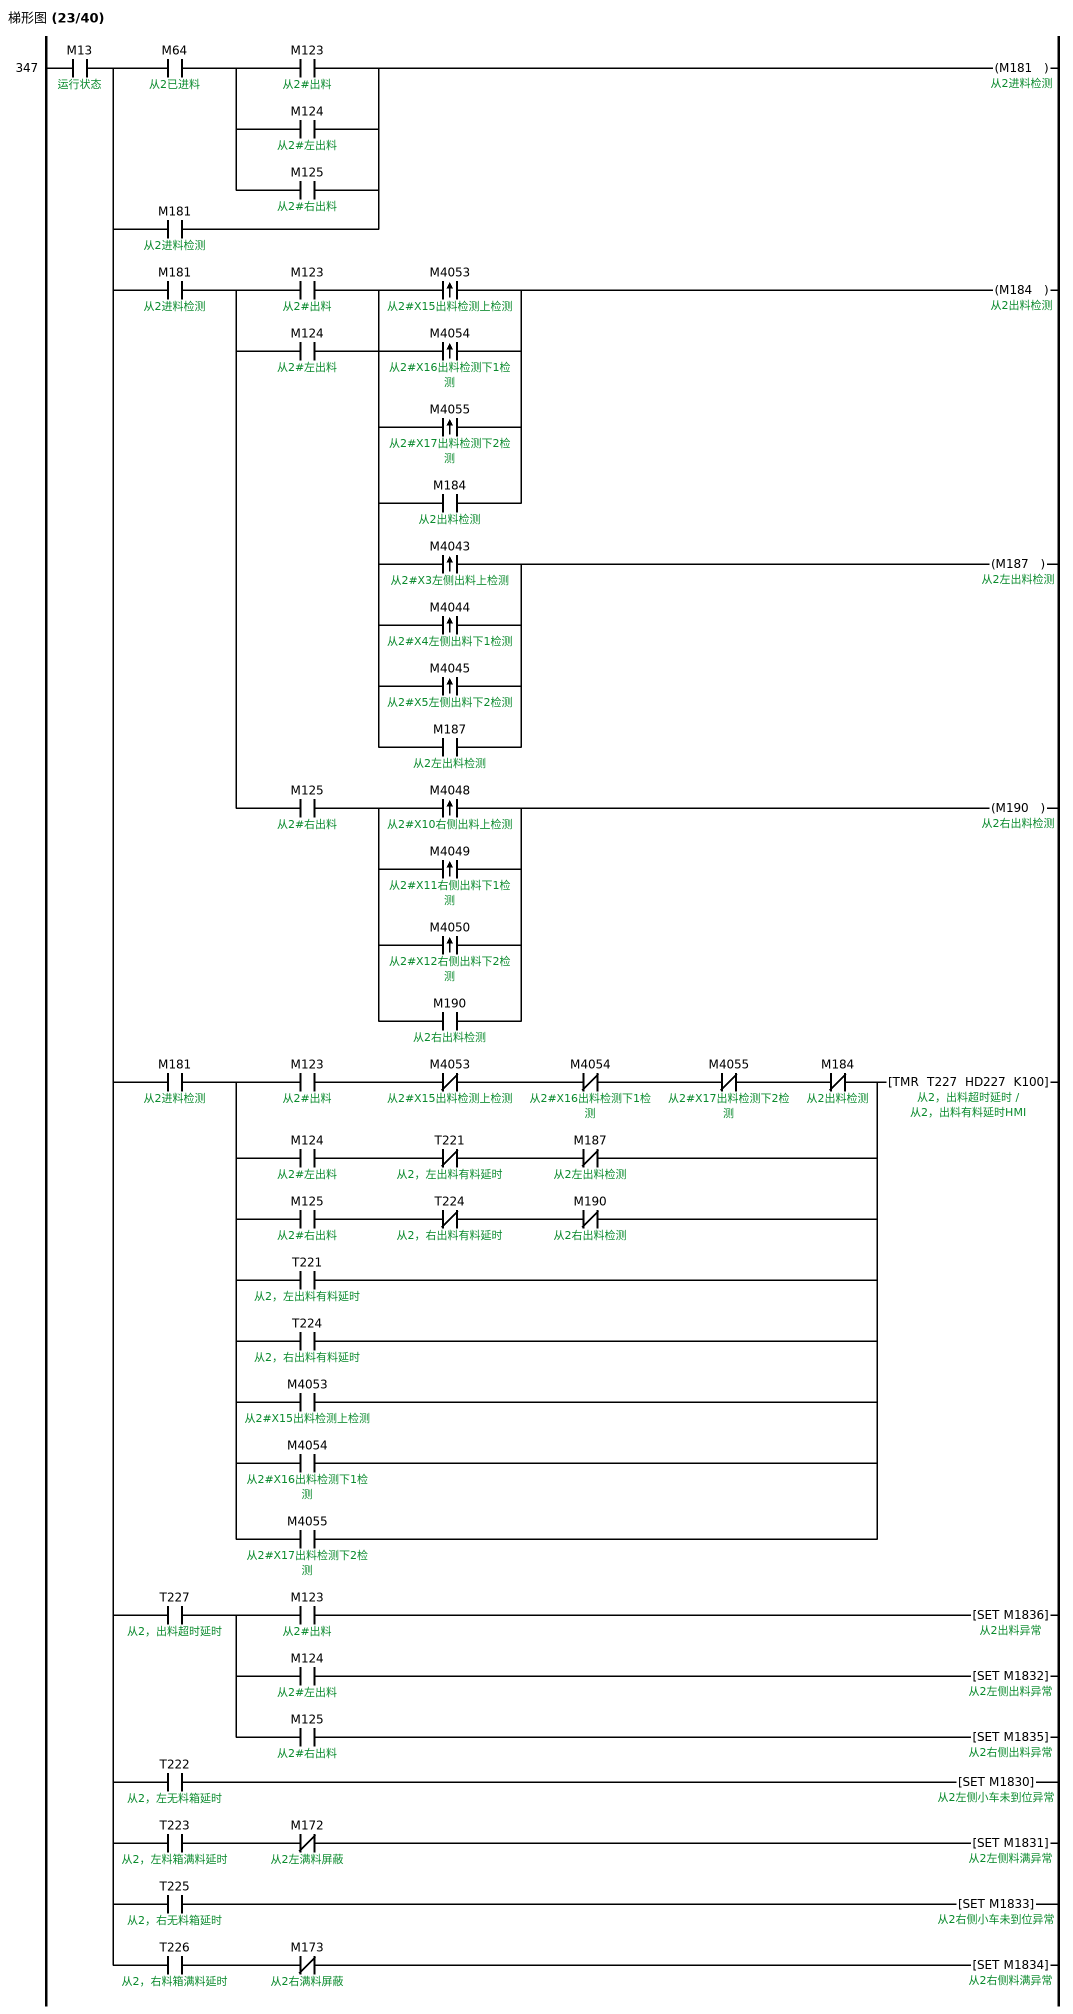
LD     M13	; 运行状态
MPS
LD     M64	; 从2已进料
LD     M123	; 从2#出料
OR     M124	; 从2#左出料
OR     M125	; 从2#右出料
ANB
OR     M181	; 从2进料检测
ANB
OUT    M181	; 从2进料检测
MRD
AND    M181	; 从2进料检测
MPS
LD     M123	; 从2#出料
OR     M124	; 从2#左出料
ANB
MPS
LDP    M4053	; 从2#X15出料检测上检测
ORP    M4054	; 从2#X16出料检测下1检测
ORP    M4055	; 从2#X17出料检测下2检测
OR     M184	; 从2出料检测
ANB
OUT    M184	; 从2出料检测
MPP
LDP    M4043	; 从2#X3左侧出料上检测
ORP    M4044	; 从2#X4左侧出料下1检测
ORP    M4045	; 从2#X5左侧出料下2检测
OR     M187	; 从2左出料检测
ANB
OUT    M187	; 从2左出料检测
MPP
AND    M125	; 从2#右出料
LDP    M4048	; 从2#X10右侧出料上检测
ORP    M4049	; 从2#X11右侧出料下1检测
ORP    M4050	; 从2#X12右侧出料下2检测
OR     M190	; 从2右出料检测
ANB
OUT    M190	; 从2右出料检测
MRD
AND    M181	; 从2进料检测
LD     M123	; 从2#出料
ANI    M4053	; 从2#X15出料检测上检测
ANI    M4054	; 从2#X16出料检测下1检测
ANI    M4055	; 从2#X17出料检测下2检测
ANI    M184	; 从2出料检测
LD     M124	; 从2#左出料
ANI    T221	; 从2，左出料有料延时
ANI    M187	; 从2左出料检测
ORB
LD     M125	; 从2#右出料
ANI    T224	; 从2，右出料有料延时
ANI    M190	; 从2右出料检测
ORB
OR     T221	; 从2，左出料有料延时
OR     T224	; 从2，右出料有料延时
OR     M4053	; 从2#X15出料检测上检测
OR     M4054	; 从2#X16出料检测下1检测
OR     M4055	; 从2#X17出料检测下2检测
ANB
TMR    T227 HD227 K100	; 从2，出料超时延时 / 从2，出料有料延时HMI
MRD
AND    T227	; 从2，出料超时延时
MPS
AND    M123	; 从2#出料
SET    M1836	; 从2出料异常
MRD
AND    M124	; 从2#左出料
SET    M1832	; 从2左侧出料异常
MPP
AND    M125	; 从2#右出料
SET    M1835	; 从2右侧出料异常
MRD
AND    T222	; 从2，左无料箱延时
SET    M1830	; 从2左侧小车未到位异常
MRD
AND    T223	; 从2，左料箱满料延时
ANI    M172	; 从2左满料屏蔽
SET    M1831	; 从2左侧料满异常
MRD
AND    T225	; 从2，右无料箱延时
SET    M1833	; 从2右侧小车未到位异常
MPP
AND    T226	; 从2，右料箱满料延时
ANI    M173	; 从2右满料屏蔽
SET    M1834	; 从2右侧料满异常

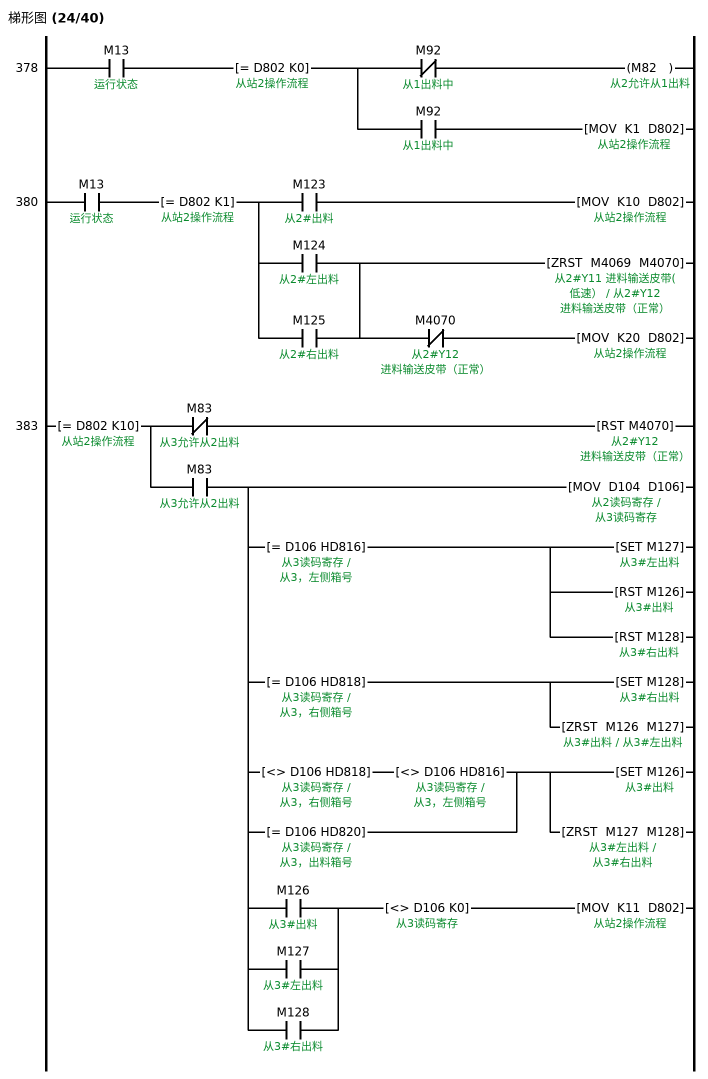
LD     M13	; 运行状态
AND=   D802 K0	; 从站2操作流程
MPS
ANI    M92	; 从1出料中
OUT    M82	; 从2允许从1出料
MPP
AND    M92	; 从1出料中
MOV    K1 D802	; 从站2操作流程
LD     M13	; 运行状态
AND=   D802 K1	; 从站2操作流程
MPS
AND    M123	; 从2#出料
MOV    K10 D802	; 从站2操作流程
MPP
LD     M124	; 从2#左出料
OR     M125	; 从2#右出料
ANB
ZRST   M4069 M4070	; 从2#Y11 进料输送皮带(低速） / 从2#Y12 进料输送皮带（正常）
ANI    M4070	; 从2#Y12 进料输送皮带（正常）
MOV    K20 D802	; 从站2操作流程
LD=    D802 K10	; 从站2操作流程
MPS
ANI    M83	; 从3允许从2出料
RST    M4070	; 从2#Y12 进料输送皮带（正常）
MPP
AND    M83	; 从3允许从2出料
MOV    D104 D106	; 从2读码寄存 / 从3读码寄存
MPS
AND=   D106 HD816	; 从3读码寄存 / 从3，左侧箱号
SET    M127	; 从3#左出料
RST    M126	; 从3#出料
RST    M128	; 从3#右出料
MRD
AND=   D106 HD818	; 从3读码寄存 / 从3，右侧箱号
SET    M128	; 从3#右出料
ZRST   M126 M127	; 从3#出料 / 从3#左出料
MRD
LD<>   D106 HD818	; 从3读码寄存 / 从3，右侧箱号
AND<>  D106 HD816	; 从3读码寄存 / 从3，左侧箱号
OR=    D106 HD820	; 从3读码寄存 / 从3，出料箱号
ANB
SET    M126	; 从3#出料
ZRST   M127 M128	; 从3#左出料 / 从3#右出料
MPP
LD     M126	; 从3#出料
OR     M127	; 从3#左出料
OR     M128	; 从3#右出料
ANB
AND<>  D106 K0	; 从3读码寄存
MOV    K11 D802	; 从站2操作流程

